FUNCTION_BLOCK WriteLRealOnlyIf
VAR_IN_OUT
	Out: LREAL;	
END_VAR
VAR_INPUT
	EN: BOOL := TRUE;
	Value: LREAL;
END_VAR
VAR_OUTPUT
	ENO: bool;
END_VAR
VAR
END_VAR

ENO := EN;
IF EN THEN
	Out := Value;
END_IF

END_FUNCTION_BLOCK

(* stored: Version 1.1.0.1, ProductVersion 3.1.4024.6
   POU WriteLRealOnlyIf: Id {095d4888-dcfd-4e6d-85cd-cff8863d336f}, SpecialFunc None *)
